// TIA Portal V20 export
ORGANIZATION_BLOCK "Startup"   // OB1030, LAD, Startup
TITLE = "Complete Restart"
// stored: AutoNumber false, Namespace Unit1.Em5, SetENOAutomatically false
   VAR_INPUT
      LostRetentive : Bool;   // True if retentive data are lost
      LostRTC : Bool;   // True if date and time are lost
   END_VAR
BEGIN

REGION Network 1 (SCL): Build the Absolut Reference Designator
   // Set the Absoult Reference Designator in the Config DB
   IF LEN(IN := "Unit1.Em5.Config".em.referenceDesignator.parent) <> 0 THEN
       "Unit1.Em5.Config".em.referenceDesignator.combined := CONCAT_WSTRING(IN1 := "Unit1.Em5.Config".em.referenceDesignator.parent, IN2 := WSTRING#'.', IN3 := "Unit1.Em5.Config".em.referenceDesignator.relative);
   ELSE
       "Unit1.Em5.Config".em.referenceDesignator.combined := "Unit1.Em5.Config".em.referenceDesignator.relative;
   END_IF;
END_REGION

REGION Network 2 (SCL): Assign axes data
   // Assign axes
   "Unit1.Em5.Config".axis[1] := "BA060AZSIDR12_TransferPnPLeftAxisX";
   "Unit1.Em5.Config".axis[2] := "BA060AZSIDR13_TransferPnPLeftAxisY";
   "Unit1.Em5.Config".axis[3] := "BA060AZSIDR14_TransferPnPLeftAxisZ";
   "Unit1.Em5.Config".axis[4] := "BA060AZSIDR15_TransferPnPRightAxisX";
   "Unit1.Em5.Config".axis[5] := "BA060AZSIDR16_TransferPnPRightAxisY";
   "Unit1.Em5.Config".axis[6] := "BA060AZSIDR17_TransferPnPRightAxisZ";

   // FB Enable
   "Unit1.Em5.HmiInterface".cmTransferPnPLeftAxisX.commands.enableMasterControl := TRUE;
   "Unit1.Em5.HmiInterface".cmTransferPnPLeftAxisY.commands.enableMasterControl := TRUE;
   "Unit1.Em5.HmiInterface".cmTransferPnPLeftAxisZ.commands.enableMasterControl := TRUE;
   "Unit1.Em5.HmiInterface".cmTransferPnPRightAxisX.commands.enableMasterControl := TRUE;
   "Unit1.Em5.HmiInterface".cmTransferPnPRightAxisY.commands.enableMasterControl := TRUE;
   "Unit1.Em5.HmiInterface".cmTransferPnPRightAxisZ.commands.enableMasterControl := TRUE;
END_REGION
END_ORGANIZATION_BLOCK
